FUNCTION AI_Scale : REAL
VAR_INPUT
	IN		:REAL;
	INmin	:REAL;
	INmax	:REAL;
	OUTmin	:REAL;
	OUTmax	:REAL;
END_VAR
VAR
	A:REAL;
	B:REAL;
END_VAR

IF IN<INmin THEN
	AI_Scale := INmin;
ELSIF IN>INmax THEN
	AI_Scale := INmax;
ELSE
	IF INmin<>INmax THEN
		A := (OUTmax-OUTmin)/(INmax-INmin);
		B := OUTmax-(A*INmax);
		AI_Scale := A*IN + B;
	END_IF
END_IF

END_FUNCTION

(* stored: Version 1.1.0.1, ProductVersion 3.1.4024.4
   POU AI_Scale: Id {b2b83a15-3659-4c8a-8335-68e4c21e2d60}, SpecialFunc None *)
